// TIA Portal V16 export
// export: Created 2024-09-05T17:39:24.0937811Z, ExportSetting WithDefaults, DisplayName Totally Integrated Automation Portal, DisplayVersion V16 Update 6, DisplayName TIA Portal Version Control Interface, DisplayVersion V16 Update 2, DisplayName TIA Portal Openness, DisplayVersion V16 Update 6, DisplayName STEP 7 Professional, DisplayVersion V16 Update 6, DisplayName STEP 7 Safety, DisplayVersion V16, DisplayName WinCC Advanced, DisplayVersion V16 Update 6
FUNCTION_BLOCK "2. Call_M000_PRODUCTION_DECLARATION"   // FB2002, LAD
{ S7_Optimized_Access := 'TRUE' }
AUTHOR : bartz
VERSION : 0.1
// stored: AutoNumber false, IsIECCheckEnabled false, IsRetainMemResEnabled false, MemoryReserve 100, SetENOAutomatically false, UDAEnableTagReadback false
   VAR_INPUT
      CYCLE_COUNTER : DInt;   // Production counter
      timeUTC { ExternalAccessible := 'False'; ExternalVisible := 'False'; ExternalWritable := 'False'} : DTL;
   END_VAR
   VAR_IN_OUT
      LOCAL_PART_ARRAY : Variant;   // Local part reference
      LOCAL_PART_WSTRING : Variant;
      LOCAL_TOOL : Variant;   // Local tool reference
      TRACA_REF : Variant;   // Traceability reference
      QUANTITY : Variant;
      STATION_NAME : Variant;
   END_VAR
   VAR
      cycleCounter_temp : DInt;
      LOCAL_PART_OK : WString;
      STATION_NAME_OK : WString;
      datestring : WString;
      READ_TIMESTAMP : DTL;
      aux : Struct
         idx : UInt;
         cnt : UInt;
         sizeCnt : Bool;
         LOCAL_PART_STRING : String;
      END_STRUCT;
   END_VAR
   VAR_TEMP
      retVal : Int;
   END_VAR
BEGIN

REGION Network 1 (SCL): PREPARE LOCAL_PART
   REGION PREPARE LOCAL_PART_ARRAY
       //Local part management - variable can be either wstring OR array of char
       IF #LOCAL_PART_WSTRING <> NULL THEN
           VariantGet(SRC := #LOCAL_PART_WSTRING,
                      DST => #LOCAL_PART_OK);
       ELSE
           IF #LOCAL_PART_ARRAY <> NULL THEN
               #aux.sizeCnt := FALSE;
               //If array of char, the array pass through a filter to delete empty positions
               Chars_TO_Strg(Chars := #LOCAL_PART_ARRAY,
                             pChars := 0,
                             Cnt := 0, //Copy all positions of char array
                             Strg => #aux.LOCAL_PART_STRING);

               //Find the last valid char
               #aux.idx := INT_TO_UINT(LEN(#aux.LOCAL_PART_STRING));

               WHILE #aux.sizeCnt = FALSE DO
                   IF #aux.LOCAL_PART_STRING[#aux.idx] <> ' ' THEN
                       //Set the index of last valid char
                       #aux.cnt := #aux.idx;
                       #aux.sizeCnt := TRUE;
                   ELSE
                       #aux.idx := #aux.idx - 1;
                   END_IF;
               END_WHILE;

               //Convert the array of char in string
               Chars_TO_Strg(Chars := #LOCAL_PART_ARRAY,
                             pChars := 0,
                             Cnt := #aux.cnt, //Copy only the right amount of data
                               Strg => #aux.LOCAL_PART_STRING);
               #LOCAL_PART_OK := STRING_TO_WSTRING(#aux.LOCAL_PART_STRING);
           ELSE
               //"MII_Parameters".M000_Status.error := TRUE;
               "MII_Parameters".M000_Status.status := WSTRING#'NO LOCAL PART DEFINED';
           END_IF;
       END_IF;
   END_REGION
END_REGION

REGION Network 2 (SCL): PREPARE CALL METHOD
   IF #cycleCounter_temp <> #CYCLE_COUNTER THEN

       IF #CYCLE_COUNTER > 0 THEN
           //Normal mode
           IF "MII_Parameters".Connection_Status.opcUaConnected THEN

               //Start attempts counter 
               "MII_Parameters".Connection_Status.aux.nAttemptsTotal := 1;

               //Set argument parameters
               "MII_Interface_Data".MII_METHODS.M000_PRODUCTION_DECLARATION.Inputs.CYCLE_COUNTER := DINT_TO_WSTRING(#CYCLE_COUNTER);
               "MII_Interface_Data".MII_METHODS.M000_PRODUCTION_DECLARATION.Inputs.LOCAL_PART := #LOCAL_PART_OK;

               // When there are more than one station at the machine, the _STn is concatenated to the PLC_ID
               IF #STATION_NAME <> NULL THEN
                   VariantGet(SRC := #STATION_NAME,
                              DST => #STATION_NAME_OK);
                   IF #STATION_NAME_OK <> WSTRING#'' THEN
                       "MII_Interface_Data".MII_METHODS.M000_PRODUCTION_DECLARATION.Inputs.PLC_ID := CONCAT_WSTRING(IN1 := "MII_Parameters".Connection.PLC_ID, IN2 := WSTRING#'_', IN3 := #STATION_NAME_OK);
                   ELSE
                       "MII_Interface_Data".MII_METHODS.M000_PRODUCTION_DECLARATION.Inputs.PLC_ID := "MII_Parameters".Connection.PLC_ID;
                   END_IF;
               ELSE
                   "MII_Interface_Data".MII_METHODS.M000_PRODUCTION_DECLARATION.Inputs.PLC_ID := "MII_Parameters".Connection.PLC_ID;
               END_IF;

               IF NOT "MII_Parameters".Connection.OperationMode THEN
                   "MII_Interface_Data".MII_METHODS.M000_PRODUCTION_DECLARATION.Inputs.PLANT := "MII_Parameters".Connection.PlantID;
               ELSE
                   "MII_Interface_Data".MII_METHODS.M000_PRODUCTION_DECLARATION.Inputs.PLANT := CONCAT(IN1 := "MII_Parameters".Connection.PlantID, IN2 := WSTRING#'_TEST');
               END_IF;

               VariantGet(SRC := #LOCAL_TOOL,
                          DST => "MII_Interface_Data".MII_METHODS.M000_PRODUCTION_DECLARATION.Inputs.LOCAL_TOOL);
               VariantGet(SRC := #TRACA_REF,
                          DST => "MII_Interface_Data".MII_METHODS.M000_PRODUCTION_DECLARATION.Inputs.TRACA_REF);
               VariantGet(SRC := #QUANTITY,
                          DST => "MII_Interface_Data".MII_METHODS.M000_PRODUCTION_DECLARATION.Inputs.QUANTITY);

               // New from version 4a
               #datestring := STRING_TO_WSTRING("LGF_DTLtoString_ISO"("date" := #timeUTC, separator := '-'));
               #datestring := REPLACE(IN1 := #datestring, IN2 := WSTRING#'T', L := 1, P := 11);
               // delete after minute
               #datestring := DELETE(IN := #datestring, L := 6, P := 24);
               "MII_Interface_Data".MII_METHODS.M000_PRODUCTION_DECLARATION.Inputs.TIMESTAMP := #datestring;

               //Set index to Production Declaration
               "1. DMC_setConnection_DB".CallBuffer[0] := TRUE;
               "MII_Parameters".M000_Status.status := WSTRING#'IN PROGRESS';

               //Store new cycle counter value
               #cycleCounter_temp := #CYCLE_COUNTER;

               //Downgraded mode - NOT USED           
          (* ELSE
               //Set argument parameters
               "MII_Parameters".M000_Status.Inputs.CYCLE_COUNTER := DINT_TO_WSTRING(#CYCLE_COUNTER);
               "MII_Parameters".M000_Status.Inputs.PLANT := "MII_Parameters".Connection.PlantID;
               "MII_Parameters".M000_Status.Inputs.PLC_ID := "MII_Parameters".Connection.PLC_ID;
               "MII_Parameters".M000_Status.Inputs.LOCAL_PART := #LOCAL_PART_OK;

               VariantGet(SRC := #LOCAL_TOOL,
                          DST => "MII_Parameters".M000_Status.Inputs.LOCAL_TOOL);
               VariantGet(SRC := #TRACA_REF,
                          DST => "MII_Parameters".M000_Status.Inputs.TRACA_REF);
               VariantGet(SRC := #QUANTITY,
                          DST => "MII_Parameters".M000_Status.Inputs.QUANTITY);

               //HMI MUST RESET THE VARIABLE AFTER STORING THE VALUES
               "MII_Parameters".M000_Status.error := TRUE;
               "MII_Parameters".M000_Status.status := Wstring#'DOWNGRADED';
               #retVal := RD_LOC_T("MII_Parameters".M000_Status.timestamp); *)
           END_IF;
       END_IF;
   END_IF;
END_REGION

REGION Network 3 (SCL): TEST MODE
   // Send pre defined data to DMC to test the communication and declaration
   IF "MII_Parameters".Commands.testProdDeclaration THEN

       //Start attempts counter 
       "MII_Parameters".Connection_Status.aux.nAttemptsTotal := 1;

       //Set standard test arguments
       "MII_Interface_Data".MII_METHODS.M000_PRODUCTION_DECLARATION.Inputs.CYCLE_COUNTER := INT_TO_WSTRING("MII_Parameters".Commands.auxTestProdDeclaration);
       "MII_Interface_Data".MII_METHODS.M000_PRODUCTION_DECLARATION.Inputs.PLANT := CONCAT(IN1 := "MII_Parameters".Connection.PlantID, IN2 := WSTRING#'_TEST');
       "MII_Interface_Data".MII_METHODS.M000_PRODUCTION_DECLARATION.Inputs.PLC_ID := "MII_Parameters".Connection.PLC_ID;
       "MII_Interface_Data".MII_METHODS.M000_PRODUCTION_DECLARATION.Inputs.LOCAL_PART := #LOCAL_PART_OK;

       // New from version 4a
       // 
       #datestring := STRING_TO_WSTRING("LGF_DTLtoString_ISO"("date" := #timeUTC, separator := '-'));
       #datestring := REPLACE(IN1 := #datestring, IN2 := WSTRING#'T', L := 1, P := 11);
       // delete after minute
       #datestring := DELETE(IN := #datestring, L := 6, P := 24);
       "MII_Interface_Data".MII_METHODS.M000_PRODUCTION_DECLARATION.Inputs.TIMESTAMP := #datestring;


       "1. DMC_setConnection_DB".CallBuffer[0] := TRUE;
       "MII_Parameters".M000_Status.status := WSTRING#'IN PROGRESS';
   END_IF;
END_REGION
END_FUNCTION_BLOCK
